FUNCTION_BLOCK TestCompositeDeep
  (* Version 1.0, 2007-05-09, Goran Cengic, Chalmers *)
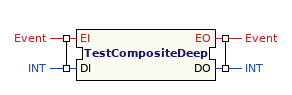
  EVENT_INPUT
    EI WITH DI;
  END_EVENT
  EVENT_OUTPUT
    EO WITH DO;
  END_EVENT
  VAR_INPUT
    DI : INT;
  END_VAR
  VAR_OUTPUT
    DO : INT;
  END_VAR
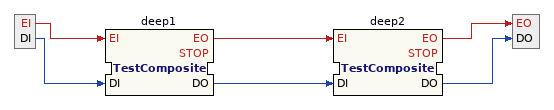
  FBS
    deep1 : TestComposite;
    deep2 : TestComposite;
  END_FBS
  EVENT_CONNECTIONS
    EI TO deep1.EI;
    deep1.EO TO deep2.EI;
    deep2.EO TO EO;
  END_CONNECTIONS
  DATA_CONNECTIONS
    DI TO deep1.DI;
    deep1.DO TO deep2.DI;
    deep2.DO TO DO;
  END_CONNECTIONS
END_FUNCTION_BLOCK
